{attribute 'GeneratedUsingTerminal: EL6720-0000-0016'}
{attribute addProperty BoxType "EL6720-0000-0016"}
{attribute addProperty Description "EL6720 Lightbus Master"}
{attribute addProperty Physics "KK"}
{attribute addProperty Id "InfoDataAT %I*InfoData_90184F0C16"}
{attribute addProperty CRC "554310285"}
{attribute addProperty Size "16"}
TYPE EL6720_210A1A8D EXTENDS EtcSlaveTerminalBase_947E5A46 :
STRUCT
	{attribute addProperty Name "InfoData"}
	InfoData : InfoData_90184F0C;
END_STRUCT
END_TYPE

(* stored: Version 1.2.0.0, ProductVersion 3.1.4024.11
   DUT EL6720_210A1A8D: Id {9f69dd80-64d5-4eec-a8ea-187e06d0dda3} *)
